(* IEC 61131-3 sources: moqui-plc/agent-skills/output/sessions/demo-plant-session/generated-plc/demo-hvac/src/main/mantle/demo-hvac, 3 files *)

(* ---- MainStatus.dut ---- *)
{attribute 'qualified_only'}
{attribute 'strict'}
TYPE MainStatus : (
    Disabled := 0,
    Standstill,
    Homing,
    Run,
    SynchronizedRun,
    Stopping,
    ErrorStop
); END_TYPE

(* Questions for the skill/user:
 * 1. Which StatusFlow is used for the main orchestration FSM?
 * 2. In which order should the states appear in the enum?
 * 3. Which state is the initial steady state?
 * 4. Which state is the fault state?
 *
 * Generation note:
 * - This enum is typically derived from StatusFlowItem entries related to the selected main StatusFlow.
 * - The generated names should match the identifiers used by Main.pou and MainRuleEngine.pou.
 *)

(* ---- Main.pou ---- *)
{attribute 'no_assign'}
(*
 * NOTE: In general, the Main component implements the control logic of automated industrial systems (Finite State Machine - FSM)
 * using hierarchical control architectures. It separates control policies from implementation mechanisms,
 * and diagnostic mechanisms from failure/error reaction and system reset policies.
 *
 * MainRuleEngine generates transition requests; Main consumes them.
 * DeviceManager orchestrates the individual device FBs.
 *
 * Call order in the PLC task:
 *   InputSignalUpdate -> Main -> DeviceManager -> OutputSignalUpdate
 *)
FUNCTION_BLOCK Main
VAR_EXTERNAL
    dev : DeviceFacade;
    workEffort : WorkEffort;
END_VAR
VAR_INPUT
    operationType : OperatingMode;
    enable : BOOL;
END_VAR
VAR_OUTPUT
    done : BOOL;
    error : BOOL;
END_VAR
VAR CONSTANT
    componentName : STRING := 'demo-hvac';
END_VAR
VAR
    (* Logger facade *)
    logger : LoggerFacade;
    (* FSM transition logic *)
    ruleEngine : MainRuleEngine;
    (* Optional: define one or more FSMs for managing subsystems, if needed *)
    (* HAL manager *)
    deviceManager : DeviceManager;
END_VAR

(* Logger facade init *)
logger.enable := TRUE; logger.loggerName := componentName;

IF NOT enable THEN RETURN; END_IF

(* Init: device setup and configuration *)
IF (operationType = OperatingMode.Init) THEN
    logger(message := 'Setup and configuration of all devices.', level := LogLevel.DEBUG);
    (* The static device configuration parameters are mapped directly by the device config manager (recipe manager),
     * while only the dynamic parameters are mapped below in the standby status.
     *)
    (* Reset signal manager *)
    dev.signalMgmt(operationType := SignalMgmtOperatingMode.Reset, loggerName := componentName);
    dev.status := MainStatus.Disabled;
    dev.lastStatus := MainStatus.Disabled;
    done := FALSE;
    dev.actualRuntime := 0;
    dev.actualBreakDuration := 0;
    dev.processActualDuration := 0;
    dev.processRemainingDuration := 0;
    dev.timeBreakEnabled := FALSE;
    dev.isCompleted := FALSE;
ELSE
    (* FSM transition-condition rule engine *)
    logger(message := 'Run FSM transition-condition logic.', level := LogLevel.DEBUG);
    ruleEngine(operationType := operationType);
END_IF;

dev.lastStatus := dev.status;

(* Fault overrides any other state *)
IF dev.faultRequest THEN dev.status := MainStatus.ErrorStop; END_IF;

(* Main FSM - Output function + State-update function *)
logger(message := 'Run Main FSM.', level := LogLevel.DEBUG);
CASE dev.status OF
    MainStatus.Disabled :
        logger(message := 'Disabled.', level := LogLevel.DEBUG);

        (* FSM output function *)
        __OUTPUT_ASSIGNMENTS_DISABLED__

        (* FSM status update function *)
        IF __COND_DISABLED_TO_STANDSTILL__ THEN
            (* Init -> Standstill *)
            dev.status := MainStatus.Standstill;
        END_IF;

    MainStatus.Standstill :
        logger(message := 'Standstill.', level := LogLevel.DEBUG);

        (* FSM output function *)
        __OUTPUT_ASSIGNMENTS_STANDSTILL__

        (* FSM status update function *)
        IF __COND_STANDSTILL_TO_HOMING__ THEN
            (* Homing -> Homing *)
            dev.status := MainStatus.Homing;
        ELSIF __COND_STANDSTILL_TO_STOPPING__ THEN
            (* Stopping -> Stopping *)
            dev.status := MainStatus.Stopping;
        ELSIF __COND_STANDSTILL_TO_RUN__ THEN
            (* Running -> Run *)
            dev.status := MainStatus.Run;
        ELSIF __COND_STANDSTILL_TO_SYNCHRONIZEDRUN__ THEN
            (* Synchronized Run -> SynchronizedRun *)
            dev.status := MainStatus.SynchronizedRun;
        ELSIF __COND_STANDSTILL_TO_ERRORSTOP__ THEN
            (* Error -> ErrorStop *)
            dev.status := MainStatus.ErrorStop;
        ELSIF __COND_STANDSTILL_TO_DISABLED__ THEN
            (* Disabling -> Disabled *)
            dev.status := MainStatus.Disabled;
        END_IF;

    MainStatus.Homing :
        logger(message := 'Homing.', level := LogLevel.DEBUG);

        (* FSM output function *)
        __OUTPUT_ASSIGNMENTS_HOMING__

        (* FSM status update function *)
        IF __COND_HOMING_TO_STANDSTILL__ THEN
            (* Standstill -> Standstill *)
            dev.status := MainStatus.Standstill;
        ELSIF __COND_HOMING_TO_STOPPING__ THEN
            (* Stopping -> Stopping *)
            dev.status := MainStatus.Stopping;
        ELSIF __COND_HOMING_TO_ERRORSTOP__ THEN
            (* Error -> ErrorStop *)
            dev.status := MainStatus.ErrorStop;
        ELSIF __COND_HOMING_TO_DISABLED__ THEN
            (* Disabling -> Disabled *)
            dev.status := MainStatus.Disabled;
        END_IF;

    MainStatus.Run :
        logger(message := 'Run.', level := LogLevel.DEBUG);

        (* FSM output function *)
        __OUTPUT_ASSIGNMENTS_RUN__

        (* FSM status update function *)
        IF __COND_RUN_TO_STANDSTILL__ THEN
            (* Standstill -> Standstill *)
            dev.status := MainStatus.Standstill;
        ELSIF __COND_RUN_TO_STOPPING__ THEN
            (* Stopping -> Stopping *)
            dev.status := MainStatus.Stopping;
        ELSIF __COND_RUN_TO_SYNCHRONIZEDRUN__ THEN
            (* Synchronized Run -> SynchronizedRun *)
            dev.status := MainStatus.SynchronizedRun;
        ELSIF __COND_RUN_TO_ERRORSTOP__ THEN
            (* Error -> ErrorStop *)
            dev.status := MainStatus.ErrorStop;
        ELSIF __COND_RUN_TO_DISABLED__ THEN
            (* Disabling -> Disabled *)
            dev.status := MainStatus.Disabled;
        END_IF;

    MainStatus.SynchronizedRun :
        logger(message := 'SynchronizedRun.', level := LogLevel.DEBUG);

        (* FSM output function *)
        __OUTPUT_ASSIGNMENTS_SYNCHRONIZEDRUN__

        (* FSM status update function *)
        IF __COND_SYNCHRONIZEDRUN_TO_STOPPING__ THEN
            (* Stopping -> Stopping *)
            dev.status := MainStatus.Stopping;
        ELSIF __COND_SYNCHRONIZEDRUN_TO_RUN__ THEN
            (* Run -> Run *)
            dev.status := MainStatus.Run;
        ELSIF __COND_SYNCHRONIZEDRUN_TO_ERRORSTOP__ THEN
            (* Error -> ErrorStop *)
            dev.status := MainStatus.ErrorStop;
        ELSIF __COND_SYNCHRONIZEDRUN_TO_DISABLED__ THEN
            (* Disabling -> Disabled *)
            dev.status := MainStatus.Disabled;
        END_IF;

    MainStatus.Stopping :
        logger(message := 'Stopping.', level := LogLevel.DEBUG);

        (* FSM output function *)
        __OUTPUT_ASSIGNMENTS_STOPPING__

        (* FSM status update function *)
        IF __COND_STOPPING_TO_STANDSTILL__ THEN
            (* Standstill -> Standstill *)
            dev.status := MainStatus.Standstill;
        ELSIF __COND_STOPPING_TO_ERRORSTOP__ THEN
            (* Error -> ErrorStop *)
            dev.status := MainStatus.ErrorStop;
        ELSIF __COND_STOPPING_TO_DISABLED__ THEN
            (* Disabling -> Disabled *)
            dev.status := MainStatus.Disabled;
        END_IF;

    MainStatus.ErrorStop :
        logger(message := 'ErrorStop.', level := LogLevel.DEBUG);

        (* FSM output function *)
        __OUTPUT_ASSIGNMENTS_ERRORSTOP__

        (* FSM status update function *)
        IF __COND_ERRORSTOP_TO_STANDSTILL__ THEN
            (* Standstill -> Standstill *)
            dev.status := MainStatus.Standstill;
        ELSIF __COND_ERRORSTOP_TO_DISABLED__ THEN
            (* Disabling -> Disabled *)
            dev.status := MainStatus.Disabled;
        END_IF;
END_CASE;

done := dev.isCompleted;

(* Device orchestration (HAL) *)
logger(message := 'Update devices.', level := LogLevel.DEBUG);
deviceManager(operationType := operationType);

(* Questions for the skill/user:
 * 1. Which StatusFlow drives this Main FSM?
 * 2. What is the initial state and what is the fault state?
 * 3. For each state, which output requests must be asserted or cleared?
 * 4. For each state, which next-state requests may be consumed here?
 *)

(* ---- MainRuleEngine.pou ---- *)
{attribute 'no_assign'}
(*
 * MainRuleEngine - transition-condition logic for the supervisor FSM.
 *
 * Responsibilities:
 *   1. Reset transition requests to safe defaults.
 *   2. Run the signal management engine (fault / alarm / warning detection).
 *   3. Compute boolean predicates from sensor feedback and recipe setpoints.
 *   4. Implement the per-state transition-condition rules.
 *
 * Default / persistence convention
 * At the top of every scan standbyRequest is set TRUE (safe default).
 * Each ACTIVE-state CASE block MUST:
 *   - Set standbyRequest := FALSE (keep current state) in the ELSE branch.
 *   - Set standbyRequest := TRUE (or leave as-is) when an EXIT condition is met.
 *   - Set standbyRequest := FALSE and another*Request := TRUE to switch phase.
 *
 * Without the ELSE branch the system would exit any active state to Standby
 * on the very first scan - a single-scan flash rather than a persistent phase.
 *)
FUNCTION_BLOCK MainRuleEngine
VAR_EXTERNAL
    clks : Clocks;
    dev : DeviceFacade;
    workEffort : WorkEffort;
END_VAR
VAR_INPUT
    operationType : OperatingMode := OperatingMode.Run;
END_VAR
VAR_OUTPUT
    error : BOOL;
END_VAR
VAR
    (* Device diagnostics *)
    deviceDiags : DeviceDiagnostics;
END_VAR

(* Reset transition requests to safe defaults.
 *
 * standbyRequest = TRUE  -> return to / stay in Standby (safe default).
 * Active-state CASE blocks override to FALSE to keep the current phase alive,
 * or set another *Request to switch phases.
 *)
dev.faultRequest := FALSE;
dev.standstillRequest := TRUE;
dev.disabledRequest := FALSE;
dev.homingRequest := FALSE;
dev.runRequest := FALSE;
dev.synchronizedRunRequest := FALSE;
dev.stoppingRequest := FALSE;
dev.errorStopRequest := FALSE;

deviceDiags(operationType := operationType, error => error);

(* Compute sensor predicates *)
(* TODO: generate or confirm process/environment/safety predicates *)

(* Process timing - generic run / break cycle *)
IF clks.clock1s THEN
    dev.processActualDuration := dev.processActualDuration + 1;

    IF dev.timeBreakEnabled AND dev.status = MainStatus.Standstill THEN
        dev.actualBreakDuration := dev.actualBreakDuration + 1;
        IF dev.estimatedBreakDuration > 0 THEN
            IF (dev.actualBreakDuration >= dev.estimatedBreakDuration)
                    AND (dev.actualBreakDuration >= dev.minBreakDuration) THEN
                dev.timeBreakEnabled := FALSE;
                dev.actualRuntime := 0;
                dev.actualBreakDuration := 0;
            END_IF;
        END_IF;
    ELSE
        dev.actualRuntime := dev.actualRuntime + 1;
        IF dev.estimatedRuntime > 0 THEN
            dev.processRemainingDuration := dev.processEstimatedDuration - dev.processActualDuration;
            IF NOT dev.timeBreakEnabled
                    AND (dev.actualRuntime >= dev.estimatedRuntime)
                    AND (dev.actualRuntime >= dev.minRuntime) THEN
                dev.timeBreakEnabled := TRUE;
                dev.actualBreakDuration := 0;
            END_IF;
        END_IF;
    END_IF;

    IF dev.processEstimatedDuration > 0 THEN
        dev.isCompleted :=
            (dev.processActualDuration >= dev.processEstimatedDuration)
            AND (dev.processActualDuration >= dev.processMinDuration);
    END_IF;
END_IF;

(* Fault gate *)
IF error OR ((dev.signalMgmt.cumulativeOutputAction AND SignalOutputAction.ImmediateStop) <> 0) THEN
    dev.faultRequest := TRUE;
    RETURN;
END_IF;

(* Transition-condition rule engine
 *
 * Persistence rule: every active-state CASE MUST end with
 *   ELSE dev.standbyRequest := FALSE; (* keep current state alive *)
 * to prevent the scan-level default (standbyRequest=TRUE) from immediately
 * bouncing the FSM back to Standby before the exit condition is reached.
 *)
CASE dev.status OF
    MainStatus.Disabled :
        (* State Disabled transition conditions *)
        IF __COND_DISABLED_TO_STANDSTILL__ THEN
            (* Init -> Standstill *)
            __ASSIGN_DISABLED_TO_STANDSTILL__
        ELSE
            dev.standstillRequest := FALSE; (* keep current state alive *)
        END_IF;

    MainStatus.Standstill :
        (* State Standstill transition conditions *)
        IF __COND_STANDSTILL_TO_HOMING__ THEN
            (* Homing -> Homing *)
            __ASSIGN_STANDSTILL_TO_HOMING__
        ELSIF __COND_STANDSTILL_TO_STOPPING__ THEN
            (* Stopping -> Stopping *)
            __ASSIGN_STANDSTILL_TO_STOPPING__
        ELSIF __COND_STANDSTILL_TO_RUN__ THEN
            (* Running -> Run *)
            __ASSIGN_STANDSTILL_TO_RUN__
        ELSIF __COND_STANDSTILL_TO_SYNCHRONIZEDRUN__ THEN
            (* Synchronized Run -> SynchronizedRun *)
            __ASSIGN_STANDSTILL_TO_SYNCHRONIZEDRUN__
        ELSIF __COND_STANDSTILL_TO_ERRORSTOP__ THEN
            (* Error -> ErrorStop *)
            __ASSIGN_STANDSTILL_TO_ERRORSTOP__
        ELSIF __COND_STANDSTILL_TO_DISABLED__ THEN
            (* Disabling -> Disabled *)
            __ASSIGN_STANDSTILL_TO_DISABLED__
        ELSE
            dev.standstillRequest := FALSE; (* keep current state alive *)
        END_IF;

    MainStatus.Homing :
        (* State Homing transition conditions *)
        IF __COND_HOMING_TO_STANDSTILL__ THEN
            (* Standstill -> Standstill *)
            __ASSIGN_HOMING_TO_STANDSTILL__
        ELSIF __COND_HOMING_TO_STOPPING__ THEN
            (* Stopping -> Stopping *)
            __ASSIGN_HOMING_TO_STOPPING__
        ELSIF __COND_HOMING_TO_ERRORSTOP__ THEN
            (* Error -> ErrorStop *)
            __ASSIGN_HOMING_TO_ERRORSTOP__
        ELSIF __COND_HOMING_TO_DISABLED__ THEN
            (* Disabling -> Disabled *)
            __ASSIGN_HOMING_TO_DISABLED__
        ELSE
            dev.standstillRequest := FALSE; (* keep current state alive *)
        END_IF;

    MainStatus.Run :
        (* State Run transition conditions *)
        IF __COND_RUN_TO_STANDSTILL__ THEN
            (* Standstill -> Standstill *)
            __ASSIGN_RUN_TO_STANDSTILL__
        ELSIF __COND_RUN_TO_STOPPING__ THEN
            (* Stopping -> Stopping *)
            __ASSIGN_RUN_TO_STOPPING__
        ELSIF __COND_RUN_TO_SYNCHRONIZEDRUN__ THEN
            (* Synchronized Run -> SynchronizedRun *)
            __ASSIGN_RUN_TO_SYNCHRONIZEDRUN__
        ELSIF __COND_RUN_TO_ERRORSTOP__ THEN
            (* Error -> ErrorStop *)
            __ASSIGN_RUN_TO_ERRORSTOP__
        ELSIF __COND_RUN_TO_DISABLED__ THEN
            (* Disabling -> Disabled *)
            __ASSIGN_RUN_TO_DISABLED__
        ELSE
            dev.standstillRequest := FALSE; (* keep current state alive *)
        END_IF;

    MainStatus.SynchronizedRun :
        (* State SynchronizedRun transition conditions *)
        IF __COND_SYNCHRONIZEDRUN_TO_STOPPING__ THEN
            (* Stopping -> Stopping *)
            __ASSIGN_SYNCHRONIZEDRUN_TO_STOPPING__
        ELSIF __COND_SYNCHRONIZEDRUN_TO_RUN__ THEN
            (* Run -> Run *)
            __ASSIGN_SYNCHRONIZEDRUN_TO_RUN__
        ELSIF __COND_SYNCHRONIZEDRUN_TO_ERRORSTOP__ THEN
            (* Error -> ErrorStop *)
            __ASSIGN_SYNCHRONIZEDRUN_TO_ERRORSTOP__
        ELSIF __COND_SYNCHRONIZEDRUN_TO_DISABLED__ THEN
            (* Disabling -> Disabled *)
            __ASSIGN_SYNCHRONIZEDRUN_TO_DISABLED__
        ELSE
            dev.standstillRequest := FALSE; (* keep current state alive *)
        END_IF;

    MainStatus.Stopping :
        (* State Stopping transition conditions *)
        IF __COND_STOPPING_TO_STANDSTILL__ THEN
            (* Standstill -> Standstill *)
            __ASSIGN_STOPPING_TO_STANDSTILL__
        ELSIF __COND_STOPPING_TO_ERRORSTOP__ THEN
            (* Error -> ErrorStop *)
            __ASSIGN_STOPPING_TO_ERRORSTOP__
        ELSIF __COND_STOPPING_TO_DISABLED__ THEN
            (* Disabling -> Disabled *)
            __ASSIGN_STOPPING_TO_DISABLED__
        ELSE
            dev.standstillRequest := FALSE; (* keep current state alive *)
        END_IF;

    MainStatus.ErrorStop :
        (* State ErrorStop transition conditions *)
        IF __COND_ERRORSTOP_TO_STANDSTILL__ THEN
            (* Standstill -> Standstill *)
            __ASSIGN_ERRORSTOP_TO_STANDSTILL__
        ELSIF __COND_ERRORSTOP_TO_DISABLED__ THEN
            (* Disabling -> Disabled *)
            __ASSIGN_ERRORSTOP_TO_DISABLED__
        ELSE
            dev.standstillRequest := FALSE; (* keep current state alive *)
        END_IF;
END_CASE;

(* Questions for the skill/user:
 * 1. Which predicates must be computed from analog/digital signals?
 * 2. Which predicates are process predicates and which are safety predicates?
 * 3. Which predicates can be inferred from existing parameter names, thresholds, hysteresis values, or seed-data rows?
 * 4. For each StatusFlowTransition, what is the boolean condition from current state to next state?
 * 5. Which transition has precedence if multiple conditions are true?
 * 6. Is the generic run/break timing block valid as-is, or does it require extension?
 *)
